// TwinCAT 3 PLC project TcpIp_CLIENT_with_TLS_PSK
// Title: TLS Sample
// Company: Beckhoff Automation
// ProjectVersion: 1.0.0.0
// ProgramVersion: 3.1.0.5
// libraries:
//   Tc2_Standard, * (Beckhoff Automation GmbH)
//   Tc2_System, * (Beckhoff Automation GmbH)
//   Tc2_TcpIp, * (Beckhoff Automation GmbH)
//   Tc2_Utilities, * (Beckhoff Automation GmbH)
//   Tc3_Module, * (Beckhoff Automation GmbH)
// project tree:
//   Data types/ E_ConnectionSteps.TcDUT
//   Global Variables/ Global_Variables.TcGVL
//   POUs/ FB_Client.TcPOU, FB_ClientApplication.TcPOU, FB_ClientConnection.TcPOU, MAIN.TcPOU
//   POUs/Helper POUs/ FB_FrameFifo.TcPOU, FB_LogFifo.TcPOU, FB_TlsConfig.TcPOU
//   / PlcTaskClient.TcTTO (not stored)
// real-time tasks:
//   TASK PlcTaskClient: cycle T#10ms, priority 21, ADS port 350

// ---- Data types/E_ConnectionSteps.TcDUT
TYPE E_ConnectionSteps :
(
	eCONNECTION_STATE_IDLE,
	eCONNECTION_STATE_SOCKET_CREATE,
	eCONNECTION_STATE_CONNECT_START,
	eCONNECTION_STATE_CONNECT_WAIT,
	eCONNECTION_STATE_DATAEXCHANGE,
	eCONNECTION_STATE_CLOSE_START,
	eCONNECTION_STATE_CLOSE_WAIT,
	eCONNECTION_STATE_ERROR
);
END_TYPE

// ---- Global Variables/Global_Variables.TcGVL
VAR_GLOBAL CONSTANT
	PLCPRJ_BUFFER_SIZE						: UDINT := 1000;

	PLCPRJ_SEND_CYCLE_TIME					: TIME := T#1S;
	PLCPRJ_RECEIVE_POLLING_TIME		 		: TIME := T#100MS;
	PLCPRJ_RECEIVE_TIMEOUT					: TIME := T#50S;

	(* Some project specific error codes *)
	PLCPRJ_ERROR_RECEIVE_TIMEOUT			: UDINT := 16#8101;(* Receive timeout error *)
	PLCPRJ_ERROR_SENDFIFO_OVERFLOW			: UDINT := 16#8102;(* Send fifo overflow *)
	PLCPRJ_ERROR_RECFIFO_OVERFLOW			: UDINT := 16#8103;(* Receive fifo overflow *)
END_VAR

// ---- POUs/FB_Client.TcPOU
FUNCTION_BLOCK FB_Client
VAR_IN_OUT
	fbTls         : FB_TlsConfig;(* TLS/PSK configuration *)
END_VAR
VAR_INPUT
	sSrvNetID     : T_AmsNetID :='';(* TwinCAT TCP/IP server network address *)
	sRemoteHost   : T_IPv4Addr :='';(* Server network address *)
	nRemotePort   : UINT       :=0;(* Server port number *)
	bEnable       : BOOL       :=FALSE;(* TRUE => enable client data exchange, FALSE => disable *)
	bLog          : BOOL       :=FALSE;(* TRUE => Enable log message output, FALSE => Disable *)
	sPrefix       : STRING     :='CLIENT::';(* Log message description string (allows the identification of log message source) *)
END_VAR
VAR_OUTPUT
	bConnected    : BOOL       := FALSE;(* TCP/IP connection state *)
END_VAR
VAR
	fbApplication : FB_ClientApplication;(* Client application control function block *)
	fbConnection  : FB_ClientConnection;(* Client connection/data exchange control function block *)
	fbTx          : FB_FrameFifo;(* Tx fifo *)
	fbRx          : FB_FrameFifo;(* Rx fifo *)
	fbLog         : FB_LogFifo;(* Log/debug/error fifo *)
END_VAR

(*-------------------------- Trigger data exchange -----------------------------------------------*)
fbConnection(sSrvNetID:=sSrvNetID, fbTls:=fbTls, fbTx:=fbTx, fbRx:=fbRx, fbLog:=fbLog,
			bEnable:=bEnable, sRemoteHost:=sRemoteHost, nRemotePort:=nRemotePort,
			bLog:=bLog, sPrefix:=sPrefix, bConnected=>bConnected);
IF fbConnection.bConnected THEN(* Connection established *)
	fbApplication(fbTx:=fbTx, fbRx:=fbRx, fbLog:=fbLog);
END_IF

END_FUNCTION_BLOCK

// ---- POUs/Helper POUs/FB_TlsConfig.TcPOU
(* TLS/PSK configuration *)
{attribute 'no_explicit_call':='Direct call not allowed for type FB_TlsConfig'}
{attribute 'no_assign'}
FUNCTION_BLOCK FB_TlsConfig
VAR
	_pskKey       : ARRAY[0..TCPADS_TLS_MAX_PSK_KEY_SIZE] OF BYTE;
	_pskKeyLen    : UDINT:=0;
	_sIdentity    : STRING(TCPADS_TLS_PSK_IDENTITY_SIZE);
	_sCaPath      : STRING(TCPADS_TLS_CERTIFICATE_PATH_SIZE);
	_sCrlPath     : STRING(TCPADS_TLS_CERTIFICATE_PATH_SIZE);
	_sCertPath    : STRING(TCPADS_TLS_CERTIFICATE_PATH_SIZE);
	_sKeyPath     : STRING(TCPADS_TLS_CERTIFICATE_PATH_SIZE);
	_sKeyPwd      : STRING(TCPADS_TLS_KEY_PASSWORD_SIZE);
	_listenFlags  : ST_TlsListenFlags:=DEFAULT_TLSLISTENFLAGS;
	_connectFlags : ST_TlsConnectFlags:=DEFAULT_TLSCONNECTFLAGS;
END_VAR

(* Adds CA certificate path *)
METHOD FINAL AddCa
VAR_INPUT
	sCaPath : STRING(TCPADS_TLS_CERTIFICATE_PATH_SIZE);
END_VAR
_sCaPath:=sCaPath;
END_METHOD

(* Adds certificate path *)
METHOD FINAL AddCert
VAR_INPUT
	sCertPath: STRING(TCPADS_TLS_CERTIFICATE_PATH_SIZE);
	sKeyPath: STRING(TCPADS_TLS_CERTIFICATE_PATH_SIZE);
	sKeyPwd: STRING(TCPADS_TLS_KEY_PASSWORD_SIZE);
END_VAR
_sCertPath:=sCertPath;
_sKeyPath:=sKeyPath;
_sKeyPwd:=sKeyPwd;
END_METHOD

METHOD FINAL AddConnectFlags
VAR_INPUT
	flags : ST_TlsConnectFlags;
END_VAR
_connectFlags:=flags;
END_METHOD

(* Adds certificate revocation list path *)
METHOD FINAL AddCrl
VAR_INPUT
	sCrlPath : STRING(TCPADS_TLS_CERTIFICATE_PATH_SIZE);
END_VAR
_sCrlPath:=sCrlPath;
END_METHOD

METHOD FINAL AddListenFlags
VAR_INPUT
	flags : ST_TlsListenFlags;
END_VAR
_listenFlags:=flags;
END_METHOD

(* Adds PSK and PSK identity *)
METHOD FINAL AddPsk
VAR_IN_OUT
	key : ARRAY[*] OF BYTE;
END_VAR
VAR_INPUT
	sIdentity : STRING(TCPADS_TLS_PSK_IDENTITY_SIZE);
END_VAR
_pskKeyLen:=MIN(DINT_TO_UDINT(UPPER_BOUND(key, 1) - LOWER_BOUND(key, 1) + 1), TCPADS_TLS_MAX_PSK_KEY_SIZE, SIZEOF(_pskKey));
MEMCPY(ADR(_pskKey[0]), ADR(key[LOWER_BOUND(key, 1)]), _pskKeyLen);
_sIdentity:=sIdentity;
END_METHOD

METHOD FINAL Clear
_sIdentity:='';
_pskKeyLen:=0;
MEMSET(ADR(_pskKey[0]), 0, SIZEOF(_pskKey));
_sCaPath:='';
_sCertPath:='';
_sKeyPath:='';
_sKeyPwd:='';
_sCrlPath:='';
_listenFlags:=DEFAULT_TLSLISTENFLAGS;
_connectFlags:=DEFAULT_TLSCONNECTFLAGS;
END_METHOD

PROPERTY FINAL connectFlags : ST_TlsConnectFlags
GET
connectFlags:=_connectFlags;
END_GET
END_PROPERTY

PROPERTY FINAL listenFlags : ST_TlsListenFlags
GET
listenFlags:=_listenFlags;
END_GET
END_PROPERTY

(* Pointer to first PSK key byte *)
PROPERTY FINAL pskKey : PVOID
GET
pskKey:=SEL(_pskKeyLen = 0, ADR(_pskKey[0]), 0);
END_GET
END_PROPERTY

(* Byte size of PSK key *)
PROPERTY FINAL pskKeyLen : UDINT(0..TCPADS_TLS_MAX_PSK_KEY_SIZE)
GET
pskKeyLen:=_pskKeyLen;
END_GET
END_PROPERTY

(* CA certificate path *)
PROPERTY FINAL sCaPath : STRING(TCPADS_TLS_CERTIFICATE_PATH_SIZE)
GET
sCaPath:=_sCaPath;
END_GET
END_PROPERTY

(* Certificate path *)
PROPERTY FINAL sCertPath : STRING(TCPADS_TLS_CERTIFICATE_PATH_SIZE)
GET
sCertPath:=_sCertPath;
END_GET
END_PROPERTY

(* Certificate revocation list path *)
PROPERTY FINAL sCrlPath : STRING(TCPADS_TLS_CERTIFICATE_PATH_SIZE)
GET
sCrlPath:=_sCrlPath;
END_GET
END_PROPERTY

(* PSK key identity *)
PROPERTY FINAL sIdentity : STRING(TCPADS_TLS_PSK_IDENTITY_SIZE)
GET
sIdentity:=_sIdentity;
END_GET
END_PROPERTY

(* Certificate key path *)
PROPERTY FINAL sKeyPath : STRING(TCPADS_TLS_CERTIFICATE_PATH_SIZE)
GET
sKeyPath:=_sKeyPath;
END_GET
END_PROPERTY

(* Certificate key password *)
PROPERTY FINAL sKeyPwd : STRING(TCPADS_TLS_KEY_PASSWORD_SIZE)
GET
sKeyPwd:=_sKeyPwd;
END_GET
END_PROPERTY

END_FUNCTION_BLOCK

// ---- POUs/FB_ClientApplication.TcPOU
(*------------- Simple TCP/IP client application. Adapt this code to match your needs. -----*)
FUNCTION_BLOCK FB_ClientApplication
VAR_IN_OUT
	fbTx        : FB_FrameFifo;(* TX fifo *)
	fbRx        : FB_FrameFifo;(* RX fifo *)
	fbLog       : FB_LogFifo;(* Log message fifo *)
END_VAR
VAR
	sToServer   : T_MaxString:='';
	sFromServer : T_MaxString:='';
	sLogMessage : T_MaxString:='';
	nCounter    : UDINT;
	fbSndTimer  : TON;
END_VAR

(*------------------- Send cyclic message strings ------------------------------------*)
fbSndTimer( IN := TRUE, PT := PLCPRJ_SEND_CYCLE_TIME );
IF fbSndTimer.Q THEN(* Send string to server *)
	fbSndTimer( IN := FALSE );

	nCounter := nCounter  + 1;
	sToServer := CONCAT( 'Client message: ', UDINT_TO_STRING(nCounter) );

	fbTx.AddTail( sPut := sToServer );(* Put string to the tx fifo *)
	IF NOT fbTx.bOk THEN(* TX fifo overflow => log error *)
		fbLog.Error( sMessage := 'FB_FrameFifo(sender)', nErrID := PLCPRJ_ERROR_SENDFIFO_OVERFLOW );
	END_IF

END_IF

(*--------------------- Get received message strings --------------------------------*)
REPEAT
	fbRx.RemoveHead( );(* Fetch string from rx fifo *)
	IF fbRx.bOk THEN(* Success *)

		(* TODO: Implement receive data handler *)
		sFromServer := fbRx.sGet;

	END_IF
UNTIL NOT fbRx.bOk
END_REPEAT

(*------------------------------- Get log/error messages from log fifo -------------*)
REPEAT
	fbLog.Remove( );
	IF fbLog.bOk THEN

		(* TODO: Implement log message handler *)
		sLogMessage := fbLog.sGet;

	END_IF
UNTIL NOT fbLog.bOk
END_REPEAT

END_FUNCTION_BLOCK

// ---- POUs/Helper POUs/FB_FrameFifo.TcPOU
(* Tx/Rx (string data) fifo control function block *)
{attribute 'no_explicit_call':='Direct call not allowed for type FB_FrameFifo'}
{attribute 'no_assign'}
FUNCTION_BLOCK FB_FrameFifo
VAR_INPUT
	bLog     : BOOL        := FALSE;(* TRUE => Enable log message output, FALSE => Disable *)
	sPrefix  : STRING      := 'Unknown::';(* Log message description string (allows the identification of log message source) *)
	sPut     : T_MaxString := ''; (* String message to add (write) to the fifo *)
END_VAR
VAR_OUTPUT
	bOk      : BOOL;(* TRUE = New entry added or removed succesfully, FALSE = Fifo overflow or fifo empty *)
	sGet     : T_MaxString := '';(* String message removed (read) from fifo *)
	nCount   : UDINT       := 0;(* Number of fifo entries *)
	cbFree   : UDINT       := 0;(* Free buffer space *)
END_VAR
VAR
	fbBuffer : FB_StringRingBuffer := (bOverwrite := FALSE);(* Basic (lower level) string buffer control function block *)
	buffer   : ARRAY[-3..PLCPRJ_BUFFER_SIZE] OF BYTE;(* Internal buffer memory *)
END_VAR

ACTION AddTail:
(* Adds new fifo entry *)
fbBuffer.A_AddTail( pBuffer:= ADR(buffer), cbBuffer:= SIZEOF(buffer),
					putValue:= sPut, bOk=>bOk, nCount=>nCount );
IF bOk THEN
	cbFree := PLCPRJ_BUFFER_SIZE - fbBuffer.cbSize;(* Calculate the free buffer space *)
	IF bLog THEN(* Log message *)
		ADSLOGSTR( ADSLOG_MSGTYPE_HINT OR ADSLOG_MSGTYPE_LOG, CONCAT( sPrefix, '"%s"' ), sPut );
	END_IF
END_IF
END_ACTION

ACTION Clear:
(* Resets fifo = clears all data *)
fbBuffer.A_Reset( pBuffer:= ADR(buffer), cbBuffer:= SIZEOF(buffer),
				bOk=>bOk, getValue=>sGet, nCount=>nCount );
cbFree := PLCPRJ_BUFFER_SIZE;(* Free buffer size *)
END_ACTION

ACTION RemoveHead:
(* Removes oldest fifo entry *)
fbBuffer.A_RemoveHead( pBuffer:= ADR(buffer), cbBuffer:= SIZEOF(buffer),
						bOk=>bOk, getValue=>sGet, nCount=>nCount );
IF bOk THEN
	cbFree := PLCPRJ_BUFFER_SIZE - fbBuffer.cbSize;(* Calculate the free buffer space *)
END_IF
END_ACTION

END_FUNCTION_BLOCK

// ---- POUs/Helper POUs/FB_LogFifo.TcPOU
(* Log/debug/error message fifo *)
{attribute 'no_explicit_call':='Direct call not allowed for type FB_LogFifo'}
{attribute 'no_assign'}
FUNCTION_BLOCK FB_LogFifo
VAR_INPUT
	bLog     : BOOL        := FALSE;(* TRUE => Enable log message output, FALSE => Disable *)
	sPrefix  : STRING      := 'Unknown::';(* Log message description string (allows the identification of log message source) *)
	
	sMessage : STRING      := '';(* String message to add (write) to the fifo *)
	nErrID   : UDINT       := 0;(* Error code to add (write) to the fifo *)
	hSocket  : T_HSOCKET;(* Socket connection handle *)
END_VAR
VAR_OUTPUT
	bOk      : BOOL;(* TRUE = New entry added or removed succesfully, FALSE = Fifo overflow or fifo empty *)
	sGet     : T_MaxString := '';(* String entry removed (read) from fifo *)
	nCount   : UDINT       := 0;(* Number of fifo entries *)
END_VAR
VAR
	fbBuffer : FB_StringRingBuffer;(* Basic (lower level) string buffer control function block *)
	buffer   : ARRAY[0..PLCPRJ_BUFFER_SIZE] OF BYTE;(* Internal buffer memory *)
	sSource  : T_MaxString;
	sPut     : T_MaxString;
END_VAR

ACTION Clear:
(* Clears all fifo entries *)
fbBuffer.A_Reset( 	pBuffer := ADR( buffer ), cbBuffer := SIZEOF( buffer ), 
					bOk=>bOk, nCount=>nCount, getValue=>sGet );
END_ACTION

ACTION Error:
(* Adds new fifo entry *)
IF nErrID = 0 THEN
	sSource := '::Error: 0x';
ELSIF ( nErrID AND 16#80000000) = 16#80000000 THEN
	IF nErrID = 16#80072746 THEN
		sSource := '::Win32 error (the connection is reset by remote side): 0x';
	ELSE
		sSource := '::Win32 error: 0x';
	END_IF
ELSIF (nErrID AND 16#00008100) = 16#00008100 THEN
	CASE nErrID OF
		PLCPRJ_ERROR_RECEIVE_TIMEOUT:
			sSource := '::PLC sample project receive timeout error: 0x';
		PLCPRJ_ERROR_SENDFIFO_OVERFLOW:
			sSource := '::PLC sample project send fifo overflow error: 0x';
		PLCPRJ_ERROR_RECFIFO_OVERFLOW:
			sSource := '::PLC sample project receive fifo overflow error: 0x';
	ELSE
		sSource := '::Other PLC sample project error: 0x';
	END_CASE
ELSIF (nErrID AND 16#00008000) = 16#00008000 THEN
	sSource := '::Internal TCP/IP Connection Server error: 0x';
ELSE
	sSource := '::TwinCAT System error: 0x';
END_IF

sPut := CONCAT( CONCAT( CONCAT( sPrefix, sMessage ), sSource ), DWORD_TO_HEXSTR( nErrID AND 16#FFFF, 0, FALSE ) ); 

fbBuffer.A_AddTail( pBuffer:= ADR(buffer), cbBuffer:= SIZEOF(buffer),
					putValue:= sPut, bOk=>bOk, nCount=>nCount );
IF bOk THEN
	IF bLog THEN(* Log error message *)
		ADSLOGSTR( ADSLOG_MSGTYPE_ERROR OR ADSLOG_MSGTYPE_LOG, '%s', sPut );	
	END_IF
END_IF
END_ACTION

ACTION Message:
(* Adds new fifo entry *)
sPut := CONCAT( CONCAT( sPrefix, sMessage ), CONCAT( '::', HSOCKET_TO_STRING(hSocket) ) );
fbBuffer.A_AddTail( pBuffer:= ADR(buffer), cbBuffer:= SIZEOF(buffer),
					putValue:= sPut, bOk=>bOk, nCount=>nCount );
IF bOk THEN
	IF bLog THEN(* Log information message *)
		ADSLOGSTR( ADSLOG_MSGTYPE_HINT OR ADSLOG_MSGTYPE_LOG, '%s', sPut );	
	END_IF
END_IF
END_ACTION

ACTION Remove:
(* Removes oldest fifo entry *)
IF nCount = 0 THEN
	sGet := '';
	bOk := FALSE;
	RETURN;
END_IF

fbBuffer.A_RemoveHead( pBuffer:= ADR(buffer), cbBuffer:= SIZEOF(buffer),
						getValue=>sGet, bOk=>bOk, nCount=>nCount );
END_ACTION

END_FUNCTION_BLOCK

// ---- POUs/FB_ClientConnection.TcPOU
FUNCTION_BLOCK FB_ClientConnection
VAR_IN_OUT
	fbTls            : FB_TlsConfig;(* TLS/PSK configuration *)
	fbTx             : FB_FrameFifo;(* TX fifo *)
	fbRx             : FB_FrameFifo;(* RX fifo *)
	fbLog            : FB_LogFifo;(* Log message fifo *)
END_VAR
VAR_INPUT
	sSrvNetID        : T_AmsNetID :='';(* TwinCAT TCP/IP server network address *)
	sRemoteHost      : T_IPv4Addr :='';(* IP adress of remote server *)
	nRemotePort      : UINT       :=0;(* Server port number *)
	bEnable          : BOOL       :=FALSE;(* TRUE => connect and exchange data, FALSE => disconnect *)
	tReconnect       : TIME       :=T#45S;(* Try to reconnect after this time *)
	bLog             : BOOL       :=FALSE;(* TRUE => Enable log message output, FALSE => Disable *)
	sPrefix          : STRING     :='CLIENT::';(* Log message description string (allows the identification of log message source) *)
END_VAR
VAR_OUTPUT
	bConnected       : BOOL       :=FALSE;(* Established connection status *)
END_VAR
VAR
	fbConnect        : FB_TlsSocketConnect;(* Connects to client socket *)
	fbClose          : FB_SocketClose;(* Closes client socket *)
	fbSend           : FB_SocketSend;(* Sends data *)
	fbReceive        : FB_SocketReceive;(* Receives data *)
	fbCreate         : FB_TlsSocketCreate:=(bListener:=FALSE);(* Creates client socket *)
	fbSetPsk         : FB_TlsSocketSetPsk;(* Configures PSK (pre-shared key) *)
	eStep            : E_ConnectionSteps;

	bSndBusy         : BOOL;(* Tx state *)
	bRcvBusy         : BOOL;(* Rx state *)
	bDisconnect      : BOOL;(* Disconnect flag, if set the socket will be closed *)
	
	fbPollTimer      : TON;(* Receive poll timer *)
	fbResponseTimer  : TON;(* Response timeout timer *)
	fbReconnectTimer : TON;(* Reconnect timer *)
	
	rxBuffer         : ARRAY[0..PLCPRJ_BUFFER_SIZE] OF BYTE;
	sTxFrame         : T_MaxString;
	sRxFrame         : T_MaxString;
	cbReceived       : UDINT;
	nLenOfString     : UDINT;(* String length inclusive the null delimiter *)
	bEndOfString     : BOOL:=FALSE;
END_VAR

CASE eStep OF
	eCONNECTION_STATE_IDLE:
		IF bEnable XOR bConnected THEN
			IF bEnable THEN
				fbReconnectTimer( IN := TRUE );
				IF fbReconnectTimer.Q THEN

					fbTx.Clear( sPrefix := CONCAT( sPrefix, 'FB_FrameFifo(sender)::' ), bLog := bLog );(* Clear send fifo *)
					fbRx.Clear( sPrefix := CONCAT( sPrefix, 'FB_FrameFifo(receiver)::' ), bLog := bLog );(* Clear receiver fifo *)
					fbLog.Clear( sPrefix := sPrefix, bLog := bLog );(* Clear log fifo *)
					bSndBusy := FALSE;
					bRcvBusy := FALSE;
					bDisconnect := FALSE;
					cbReceived := 0;

					fbPollTimer( IN := FALSE, PT := T#0S );
					fbResponseTimer( IN := FALSE, PT := PLCPRJ_RECEIVE_TIMEOUT );
					fbReconnectTimer( IN := FALSE, PT := tReconnect );

					fbCreate(bExecute:=FALSE);
					fbCreate(sSrvNetID:=sSrvNetID, bExecute:=TRUE);
					eStep := eCONNECTION_STATE_SOCKET_CREATE;
				END_IF
			ELSE
				eStep := eCONNECTION_STATE_CLOSE_START;
			END_IF
		ELSIF bConnected THEN
			eStep := eCONNECTION_STATE_DATAEXCHANGE;
		ELSE
			fbReconnectTimer( IN := FALSE, PT := T#0S );
		END_IF
		
	eCONNECTION_STATE_SOCKET_CREATE:
		fbCreate(bExecute:=FALSE);
		IF NOT fbCreate.bBusy THEN
			IF NOT fbCreate.bError THEN
				fbSetPsk(bExecute:=FALSE);
				IF (fbTls.pskKeyLen <> 0) AND (fbTls.pskKey <> 0) AND (fbTls.sIdentity <> '') THEN
					fbSetPsk(sSrvNetID:=sSrvNetID, hSocket:=fbCreate.hSocket, sIdentity:=fbTls.sIdentity, pskKey:=fbTls.pskKey, pskKeyLen:=fbTls.pskKeyLen, bExecute:=TRUE);
				END_IF
				eStep := eCONNECTION_STATE_CONNECT_START;
			ELSE
				fbLog.Error( sMessage := 'FB_TlsSocketCreate()', nErrID := fbCreate.nErrId );
				eStep := eCONNECTION_STATE_ERROR;
			END_IF
		END_IF

	eCONNECTION_STATE_CONNECT_START:
		fbSetPsk(bExecute:=FALSE);
		IF NOT fbSetPsk.bBusy THEN
			IF NOT fbSetPsk.bError THEN
				fbConnect(hSocket:=fbCreate.hSocket, bExecute:=FALSE);
				fbConnect(sSrvNetID:=sSrvNetID, hSocket:=fbCreate.hSocket, bExecute:=TRUE, sRemoteHost := sRemoteHost, nRemotePort := nRemotePort);
				eStep := eCONNECTION_STATE_CONNECT_WAIT;
			ELSE
				fbLog.Error( sMessage := 'FB_TlsSocketSetPsk()', nErrID := fbSetPsk.nErrId );
				eStep := eCONNECTION_STATE_ERROR;
			END_IF
		END_IF

	eCONNECTION_STATE_CONNECT_WAIT:
		fbConnect(hSocket:=fbCreate.hSocket, bExecute:=FALSE);
		IF NOT fbConnect.bBusy THEN
			IF NOT fbConnect.bError THEN
				bConnected 	:= TRUE;
				fbLog.Message( sMessage := 'Connection established!', hSocket := fbCreate.hSocket );
				eStep := eCONNECTION_STATE_IDLE;
			ELSE
				fbLog.Error( sMessage := 'FB_TlsSocketConnect()', nErrID := fbConnect.nErrId );
				eStep := eCONNECTION_STATE_ERROR;
			END_IF
		END_IF

	eCONNECTION_STATE_DATAEXCHANGE:

		bDisconnect := NOT bEnable OR bDisconnect;(* User/internal disconnect requested? *)
		IF bDisconnect AND NOT bSndBusy AND NOT bRcvBusy THEN
			bDisconnect := FALSE;
			eStep := eCONNECTION_STATE_CLOSE_START;(* Disconnect *)
		ELSE
	
			(* Send tx data *)
			IF NOT bDisconnect AND NOT bSndBusy THEN
				fbTx.RemoveHead( sGet => sTxFrame );(* Remove oldest string entry s*)
				IF fbTx.bOk THEN(* Success *)
					fbSend(bExecute:=FALSE);
					fbSend(sSrvNetID:=sSrvNetID, hSocket:=fbCreate.hSocket,
							pSrc:=ADR(sTxFrame),
							cbLen:=INT_TO_UDINT(LEN(sTxFrame)) + 1,(* String length inclusive the zero delimiter *)
							bExecute:= TRUE );
					bSndBusy := TRUE;
				END_IF
			ELSE
				fbSend(bExecute:=FALSE);
				IF NOT fbSend.bBusy THEN
					bSndBusy := FALSE;
					IF fbSend.bError THEN
						fbLog.Error( sMessage := 'FB_SocketSend()', nErrId := fbSend.nErrId );
						bDisconnect := TRUE;(* Set flag *)
					END_IF
				END_IF
			END_IF

			(* Get rx data *)
			IF NOT bDisconnect AND NOT bRcvBusy THEN
				fbPollTimer( IN := TRUE );
				IF fbPollTimer.Q THEN
					fbPollTimer( IN := FALSE, PT := PLCPRJ_RECEIVE_POLLING_TIME );
					fbReceive(bExecute:=FALSE);
					fbReceive(sSrvNetID:=sSrvNetID,
								hSocket:=fbCreate.hSocket,
								pDest:=ADR(rxBuffer) + cbReceived,
								cbLen:=SIZEOF(rxBuffer) - cbReceived,
								bExecute:=TRUE);
					bRcvBusy := TRUE;
				END_IF
			ELSE
				fbReceive(bExecute:=FALSE);
				IF NOT fbReceive.bBusy THEN
					bRcvBusy := FALSE;
					IF NOT fbReceive.bError THEN
						IF (fbReceive.nRecBytes > 0) THEN(* Bytes received *)
							
							fbPollTimer( IN := FALSE, PT := T#0S ); (* Bytes received => increase the read (polling) speed *)
							fbResponseTimer( IN := FALSE );(* Bytes received => disable timeout check *)
							cbReceived 	:= cbReceived + fbReceive.nRecBytes;(* Calculate the number of received data bytes *)

							REPEAT
								
								(* Search for string end delimiter *)
								nLenOfString := 0;(* Reset string length *)
								bEndOfString := FALSE;
								REPEAT 
									IF rxBuffer[nLenOfString] = 0 THEN(* String end delimiter found *)
										bEndOfString := TRUE;
									END_IF
									nLenOfString := nLenOfString + 1;
								UNTIL bEndOfString OR (nLenOfString >= cbReceived)
								END_REPEAT
								
								IF bEndOfString THEN
									MEMSET( ADR( sRxFrame ), 0, SIZEOF( sRxFrame ) );
									MEMCPY(  ADR( sRxFrame ), ADR( rxBuffer ), MIN( SIZEOF(sRxFrame), nLenOfString ) );(* Copy the received string to the output variable (inclusive the end delimiter) *)
									MEMMOVE( ADR( rxBuffer ), ADR( rxBuffer[nLenOfString] ), cbReceived - nLenOfString  );(* Move the reamaining data bytes *)
									cbReceived := cbReceived - nLenOfString;(* Recalculate the reamaining data byte length *)
			
									fbRx.AddTail( sPut := sRxFrame );(* Put received message to the rx fifo *)
									IF NOT fbRx.bOk THEN
										fbLog.Error( sMessage := 'FB_FrameFifo(receiver)', nErrID := PLCPRJ_ERROR_RECFIFO_OVERFLOW );
										bDisconnect := TRUE;(* Set flag *)
										RETURN;
									END_IF
								END_IF
								
							UNTIL NOT bEndOfString OR (cbReceived = 0)
							END_REPEAT
		
						ELSE(* No bytes received *)
							fbResponseTimer( IN := TRUE, PT := PLCPRJ_RECEIVE_TIMEOUT );(* No bytes received => enable timeout check *)
							IF fbResponseTimer.Q THEN (* Timeout error*)
								fbResponseTimer( IN := FALSE );
								fbLog.Error( sMessage := 'FB_SocketReceive()', nErrID := PLCPRJ_ERROR_RECEIVE_TIMEOUT );
								bDisconnect := TRUE;(* Set flag *)
							END_IF
						END_IF
						
					ELSE(* Receive error *)
						fbLog.Error( sMessage := 'FB_SocketReceive()', nErrId := fbReceive.nErrId );
						bDisconnect := TRUE;(* Set flag *)
					END_IF
				END_IF(* IF NOT fbReceive.bBusy THEN *)
				
			END_IF(* IF NOT bDisconnect AND NOT bRcvBusy THEN *)
		
		END_IF(* IF bDisconnect AND NOT bSndBusy AND NOT bRcvBusy THEN *)

		
	eCONNECTION_STATE_CLOSE_START:
		fbLog.Message( sMessage := 'Closing connection!', hSocket := fbCreate.hSocket );
		fbClose(bExecute:=FALSE);
		fbClose(sSrvNetID:=sSrvNetID,
				hSocket:=fbCreate.hSocket,
				bExecute:=TRUE);
		eStep := eCONNECTION_STATE_CLOSE_WAIT;

	eCONNECTION_STATE_CLOSE_WAIT:
		fbClose(bExecute:=FALSE);
		IF NOT fbClose.bBusy THEN
			bConnected := FALSE;
			IF NOT fbClose.bError THEN
				eStep := eCONNECTION_STATE_IDLE;
			ELSE
				fbLog.Error( sMessage := 'FB_SocketClose()', nErrID := fbClose.nErrId );
				eStep := eCONNECTION_STATE_ERROR;
			END_IF
		END_IF

	eCONNECTION_STATE_ERROR:(* Error step *)
		IF bConnected THEN
			eStep := eCONNECTION_STATE_CLOSE_START;
		ELSE
			eStep := eCONNECTION_STATE_IDLE;
		END_IF
END_CASE

END_FUNCTION_BLOCK

// ---- POUs/MAIN.TcPOU
PROGRAM MAIN
VAR
	sSrvNetID   : T_AmsNetID :='';(* TwinCAT TCP/IP server network address *)
	{warning 'Please configure your server IP-address and server port number below:'}
	sRemoteHost : T_IPv4Addr :='127.0.0.1';(* IP address of remote server! *)
	nRemotePort : UINT       :=200;(* Port number of remote server! *)
	bEnable1    : BOOL       :=TRUE;(* TRUE => Enable client1 data exchange, FALSE => Disable *)
	bEnable2    : BOOL       :=FALSE;(* TRUE => Enable client2 data exchange, FALSE => Disable *)
	bEnable3    : BOOL       :=FALSE;(* TRUE => Enable client3 data exchange, FALSE => Disable *)
	bEnable4    : BOOL       :=FALSE;(* TRUE => Enable client3 data exchange, FALSE => Disable *)
	bEnable5    : BOOL       :=FALSE;(* TRUE => Enable client5 data exchange, FALSE => Disable *)
	bLog        : BOOL       :=TRUE;(* TRUE => Enable message/error log, FALSE => Disable*)

	bPSK        : BOOL       :=TRUE;(* TRUE => use PSK , FALSE => don't use PSK *)
	key         : ARRAY[0..14] OF BYTE:=[16#1B,16#D0,16#6F,16#D2,16#56,16#16,16#7D,16#C1,16#E8,16#C7,16#48,16#2A,16#8E,16#F5,16#FF];
	fbTls       : FB_TlsConfig;(* TLS/PSK configuration *)

	fbClient1   : FB_Client:=(sRemoteHost:=sRemoteHost, nRemotePort:=nRemotePort, sPrefix:='CLIENT1::');(* TCP/IP client (connection) instance *)
	fbClient2   : FB_Client:=(sRemoteHost:=sRemoteHost, nRemotePort:=nRemotePort, sPrefix:='CLIENT2::');
	fbClient3   : FB_Client:=(sRemoteHost:=sRemoteHost, nRemotePort:=nRemotePort, sPrefix:='CLIENT3::');
	fbClient4   : FB_Client:=(sRemoteHost:=sRemoteHost, nRemotePort:=nRemotePort, sPrefix:='CLIENT4::');
	fbClient5   : FB_Client:=(sRemoteHost:=sRemoteHost, nRemotePort:=nRemotePort, sPrefix:='CLIENT5::');
	fbCloseAll  : FB_SocketCloseAll;
	bInitialize : BOOL:=TRUE;
END_VAR

IF bInitialize THEN
	(* On PLC reset or program download close all created/opened sockets/connections *)
	fbCloseAll(sSrvNetID:=sSrvNetID, bExecute:=bInitialize);
	IF fbCloseAll.bBusy OR fbCloseAll.bError THEN
		RETURN;
	END_IF

	(* Configure TLS/PSK settings *)
	fbTls.Clear();
	IF bPSK THEN
		fbTls.AddPsk(key:=key, sIdentity:='MyIdentity');
	END_IF

	bInitialize:=FALSE;
END_IF

fbClient1(fbTls:=fbTls, sSrvNetID:=sSrvNetID, bEnable:=bEnable1, bLog:=bLog);
fbClient2(fbTls:=fbTls, sSrvNetID:=sSrvNetID, bEnable:=bEnable2, bLog:=bLog);
fbClient3(fbTls:=fbTls, sSrvNetID:=sSrvNetID, bEnable:=bEnable3, bLog:=bLog);
fbClient4(fbTls:=fbTls, sSrvNetID:=sSrvNetID, bEnable:=bEnable4, bLog:=bLog);
fbClient5(fbTls:=fbTls, sSrvNetID:=sSrvNetID, bEnable:=bEnable5, bLog:=bLog);

END_PROGRAM
